// TIA Portal V16 export
// export: Created 2021-03-04T22:04:03.5713358Z, ExportSetting WithDefaults, DisplayName Totally Integrated Automation Portal, DisplayVersion V16, DisplayName TIA Portal Version Control Interface, DisplayVersion V16, DisplayName TIA Portal Openness, DisplayVersion V16, DisplayName SINAMICS Startdrive Advanced, DisplayVersion V16, DisplayName SINAMICS Startdrive G130, G150, S120, S150, SINAMICS MV, S210, DisplayVersion V16, DisplayName SINAMICS Startdrive G110M, G120, G120C, G120D, G120P, DisplayVersion V16, DisplayName STEP 7 Professional, DisplayVersion V16, DisplayName STEP 7 Safety, DisplayVersion V16, DisplayName WinCC Professional, DisplayVersion V16
FUNCTION "fcWordToBits" : Void   // FC303, LAD
TITLE = Breaks A Word Into Individual Bits
{ S7_Optimized_Access := 'TRUE' }
AUTHOR : DMC
FAMILY : LowLevel
VERSION : 0.1
// stored: AutoNumber false, IsIECCheckEnabled false, SetENOAutomatically false, UDAEnableTagReadback false
   VAR_INPUT
      wInWord : Word;   // Word to be broken into individual bits
   END_VAR
   VAR_OUTPUT
      bOutBit00 : Bool;   // Bit 0
      bOutBit01 : Bool;   // Bit 1
      bOutBit02 : Bool;   // Bit 2
      bOutBit03 : Bool;   // Bit 3
      bOutBit04 : Bool;   // Bit 4
      bOutBit05 : Bool;   // Bit 5
      bOutBit06 : Bool;   // Bit 6
      bOutBit07 : Bool;   // Bit 7
      bOutBit08 : Bool;   // Bit 8
      bOutBit09 : Bool;   // Bit 9
      bOutBit10 : Bool;   // Bit 10
      bOutBit11 : Bool;   // Bit 11
      bOutBit12 : Bool;   // Bit 12
      bOutBit13 : Bool;   // Bit 13
      bOutBit14 : Bool;   // Bit 14
      bOutBit15 : Bool;   // Bit 15
   END_VAR
BEGIN

REGION Network 1: Bit0
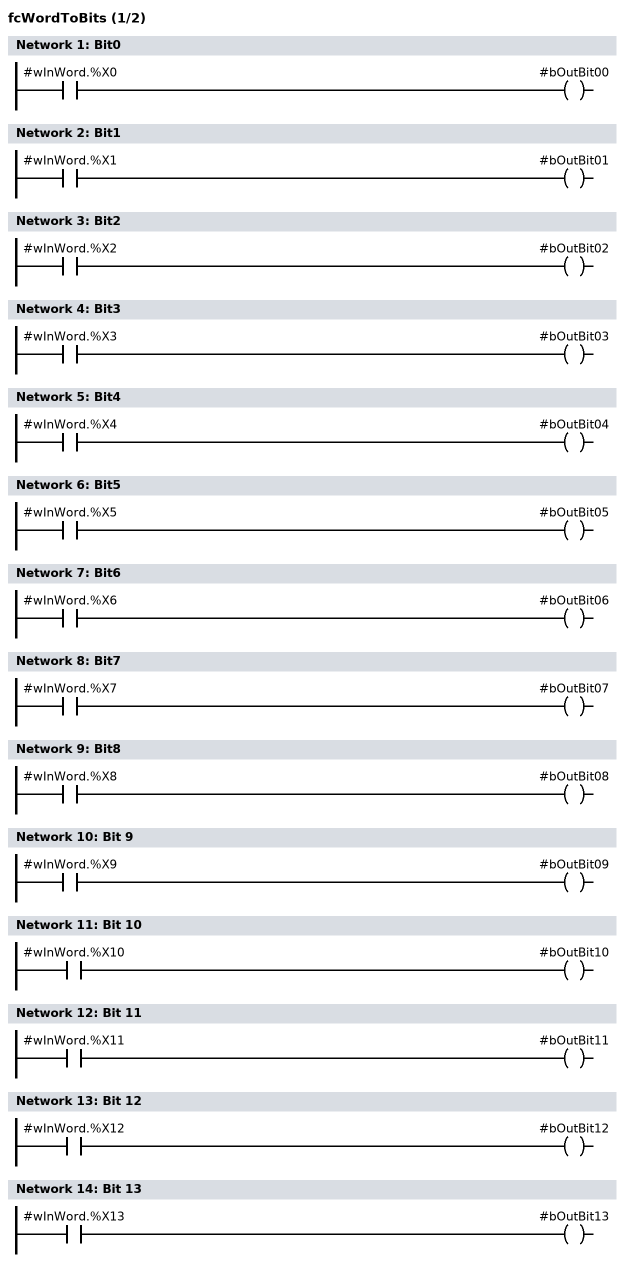
   RUNG wire#powerrail
      Contact( #wInWord.%X0 )
      Coil( #bOutBit00 )
   END_RUNG
   // the same network as SCL:
   #bOutBit00 := #wInWord.%X0;
END_REGION

REGION Network 2: Bit1
   RUNG wire#powerrail
      Contact( #wInWord.%X1 )
      Coil( #bOutBit01 )
   END_RUNG
   // the same network as SCL:
   #bOutBit01 := #wInWord.%X1;
END_REGION

REGION Network 3: Bit2
   RUNG wire#powerrail
      Contact( #wInWord.%X2 )
      Coil( #bOutBit02 )
   END_RUNG
   // the same network as SCL:
   #bOutBit02 := #wInWord.%X2;
END_REGION

REGION Network 4: Bit3
   RUNG wire#powerrail
      Contact( #wInWord.%X3 )
      Coil( #bOutBit03 )
   END_RUNG
   // the same network as SCL:
   #bOutBit03 := #wInWord.%X3;
END_REGION

REGION Network 5: Bit4
   RUNG wire#powerrail
      Contact( #wInWord.%X4 )
      Coil( #bOutBit04 )
   END_RUNG
   // the same network as SCL:
   #bOutBit04 := #wInWord.%X4;
END_REGION

REGION Network 6: Bit5
   RUNG wire#powerrail
      Contact( #wInWord.%X5 )
      Coil( #bOutBit05 )
   END_RUNG
   // the same network as SCL:
   #bOutBit05 := #wInWord.%X5;
END_REGION

REGION Network 7: Bit6
   RUNG wire#powerrail
      Contact( #wInWord.%X6 )
      Coil( #bOutBit06 )
   END_RUNG
   // the same network as SCL:
   #bOutBit06 := #wInWord.%X6;
END_REGION

REGION Network 8: Bit7
   RUNG wire#powerrail
      Contact( #wInWord.%X7 )
      Coil( #bOutBit07 )
   END_RUNG
   // the same network as SCL:
   #bOutBit07 := #wInWord.%X7;
END_REGION

REGION Network 9: Bit8
   RUNG wire#powerrail
      Contact( #wInWord.%X8 )
      Coil( #bOutBit08 )
   END_RUNG
   // the same network as SCL:
   #bOutBit08 := #wInWord.%X8;
END_REGION

REGION Network 10: Bit 9
   RUNG wire#powerrail
      Contact( #wInWord.%X9 )
      Coil( #bOutBit09 )
   END_RUNG
   // the same network as SCL:
   #bOutBit09 := #wInWord.%X9;
END_REGION

REGION Network 11: Bit 10
   RUNG wire#powerrail
      Contact( #wInWord.%X10 )
      Coil( #bOutBit10 )
   END_RUNG
   // the same network as SCL:
   #bOutBit10 := #wInWord.%X10;
END_REGION

REGION Network 12: Bit 11
   RUNG wire#powerrail
      Contact( #wInWord.%X11 )
      Coil( #bOutBit11 )
   END_RUNG
   // the same network as SCL:
   #bOutBit11 := #wInWord.%X11;
END_REGION

REGION Network 13: Bit 12
   RUNG wire#powerrail
      Contact( #wInWord.%X12 )
      Coil( #bOutBit12 )
   END_RUNG
   // the same network as SCL:
   #bOutBit12 := #wInWord.%X12;
END_REGION

REGION Network 14: Bit 13
   RUNG wire#powerrail
      Contact( #wInWord.%X13 )
      Coil( #bOutBit13 )
   END_RUNG
   // the same network as SCL:
   #bOutBit13 := #wInWord.%X13;
END_REGION

REGION Network 15: Bit 14
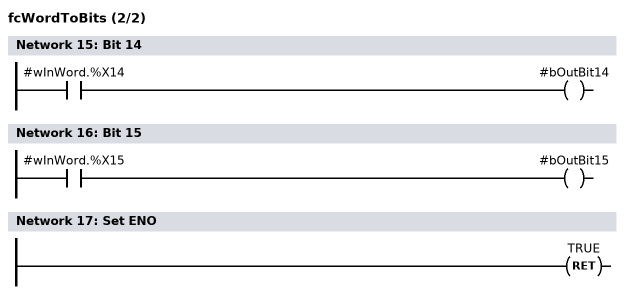
   RUNG wire#powerrail
      Contact( #wInWord.%X14 )
      Coil( #bOutBit14 )
   END_RUNG
   // the same network as SCL:
   #bOutBit14 := #wInWord.%X14;
END_REGION

REGION Network 16: Bit 15
   RUNG wire#powerrail
      Contact( #wInWord.%X15 )
      Coil( #bOutBit15 )
   END_RUNG
   // the same network as SCL:
   #bOutBit15 := #wInWord.%X15;
END_REGION

REGION Network 17: Set ENO
   RUNG wire#powerrail
      ReturnCoil( TRUE )
   END_RUNG
   // the same network as SCL:
   ENO := TRUE;
   RETURN;
END_REGION
END_FUNCTION
